{attribute 'qualified_only'}
{attribute 'strict'}
{attribute 'to_string'}
TYPE E_HE_SolidAttenuatorCommand :
(
    CALCULATE := 0
);
END_TYPE

(* stored: Version 1.1.0.1
   DUT E_HE_SolidAttenuatorCommand: Id {2f764ab7-7fa2-420e-810b-7a7ca2447215} *)
